FUNCTION_BLOCK FbDispersion (* Дисперсия PV. *)
  (* Standard: 61499-1; Description: Дисперсия PV. Simple FB with one algorithm *)
  (* Version 1.1, 2026-03-22, VA, LIB_PLC *)
  (* Documentation:
  // Дисперсия PV. //       DbDispersion //     +--------------+ //     | FbDispersion | //  ->-|In    Variance|->- //     |     Deviation|->- //     |          Mean|->- //     +--------------+
  *)
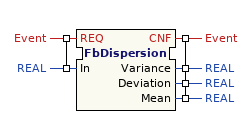
  EVENT_INPUT
    REQ WITH In; (* Normal Execution Request *)
  END_EVENT
  EVENT_OUTPUT
    CNF WITH Variance, Deviation, Mean; (* Execution Confirmation *)
  END_EVENT
  VAR_INPUT
    In : REAL := 0.0; (* Вход измерения. *)
  END_VAR
  VAR_OUTPUT
    Variance : REAL := 0.0; (* Дисперсия. *)
    Deviation : REAL := 0.0; (* Среднеквадратическое отклонение. *)
    Mean : REAL := 0.0; (* Математическое ожидание (Среднее арифметическое). *)
  END_VAR
  VAR CONSTANT
    NUMBER : INT := 99; (* Размер массива 100. *)
  END_VAR
  VAR
    Buffer1 : ARRAY [0..NUMBER] OF REAL; (* Буфер. *)
    Summator : REAL := 0.0; (* Сумматор. *)
  END_VAR
  EC_STATES
    REQ : REQ -> CNF;
  END_STATES
  ALGORITHM REQ IN ST:
VAR_TEMP
	Counter1 : INT := 0; // Счетчик.
END_VAR

// Обновление массива.
FOR Counter1 := NUMBER TO 1 BY -1 DO
	Buffer1[Counter1] := Buffer1[Counter1 - 1];
END_FOR;
Buffer1[0] := In;

// Расчет математического ожидания (среднего арифметического).
Summator := 0.0;
FOR Counter1 := 0 TO NUMBER BY 1 DO
	Summator := Summator + Buffer1[Counter1];
END_FOR;
Mean := Summator / (INT_TO_REAL(NUMBER + 1));

// Рассчет дисперсии.
Summator := 0.0;
FOR Counter1 := 0 TO NUMBER BY 1 DO
	Summator := Summator + ((Buffer1[Counter1] - Mean) * (Buffer1[Counter1] - Mean));
END_FOR;
Variance := Summator / (INT_TO_REAL(NUMBER + 1));

// Рассчет среднеквадратического отклонения.
Deviation := SQRT(Variance);

// @COPYLEFT ALL WRONGS RESERVED :)
// Author: VA
// Contacts: DIY.PLC.314@gmail.com
// Date start LIB_PLC: 2014
// License: GNU GPL-2.0-or-later
// https://www.gnu.org/licenses/old-licenses/gpl-2.0.html
// https://www.youtube.com/watch?v=n1F_MfLRlX0
// https://www.youtube.com/@DIY_PLC
// https://github.com/DIYPLC/LIB_PLC
// https://oshwlab.com/diy.plc.314/PLC_HW1_SW1
// https://3dtoday.ru/3d-models/mechanical-parts/body/korpus-na-din-reiku
// https://t.me/DIY_PLC
  END_ALGORITHM
END_FUNCTION_BLOCK
